FUNCTION_BLOCK ASEL_UINT (* Selects an element of a UINT Array *)
  (* Standard: 61499-1; Classification: Math; Function: Array element selection; Type: UINT *)
  (* Version 0.1, 2006-09-06, JHC, Holobloc Inc, Made a SimpleFB *)
  (* Version 0.0, 2005-12-13, JHC, Holobloc Inc *)
  (* Compiler header: package fb.rt.student; *)
  (* Compiler classdef: SimpleFB *)
  (* Compiler Java Sun JDK 1.5.0 *)
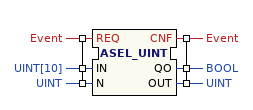
  EVENT_INPUT
    REQ WITH IN, N; (* Normal Execution Request *)
  END_EVENT
  EVENT_OUTPUT
    CNF WITH QO, OUT; (* Execution Confirmation *)
  END_EVENT
  VAR_INPUT
    IN : ARRAY [0..9] OF UINT; (* Input array *)
    N : UINT; (* Zero-based index of OUT value in IN array *)
  END_VAR
  VAR_OUTPUT
    QO : BOOL; (* OUT value validity *)
    OUT : UINT;
  END_VAR
  ALGORITHM REQ IN ST: (* Normally executed algorithm *)
IF N > 9 THEN QO := false;
ELSE
QO := true;
OUT := IN[N];
END_IF;
  END_ALGORITHM
END_FUNCTION_BLOCK
